TYPE Status_KK : (Initialisieren, Lesen, Abtauen_elektrisch, Abtauen_Heissgas_oben, Abtauen_Heissgas_unten, Vollautomatik, Manuell, Anlagenschutz, Schreiben);
END_TYPE

(* stored: Version 1.1.0.1, ProductVersion 3.1.4018.5
   DUT Status_KK: Id {9c78300b-74a9-4626-a375-a9a377526c19} *)
